// TIA Portal V17 export
// export: Created 2026-07-07T16:10:25.1870439Z, ExportSetting WithDefaults, DisplayName Totally Integrated Automation Portal, DisplayVersion V17, DisplayName TIA Portal Openness, DisplayVersion V17, DisplayName TIA Portal Version Control Interface, DisplayVersion V17, DisplayName STEP 7 Professional, DisplayVersion V17, DisplayName STEP 7 Safety, DisplayVersion V17, DisplayName WinCC Professional, DisplayVersion V17
FUNCTION_BLOCK "Manchester_Decoding"   // FB2, LAD
{ S7_Optimized_Access := 'TRUE' }
VERSION : 0.1
// stored: AutoNumber true, IsIECCheckEnabled false, IsRetainMemResEnabled false, MemoryReserve 100, SetENOAutomatically false, UDAEnableTagReadback false
   VAR_INPUT
      Clock_signal : Bool;
      Data_signal : Bool;
      "No. of inputs" : Int;
      "Interchar_duration(ms)" : Int;
   END_VAR
   VAR_OUTPUT
      Input_1 : Bool;
      Input_2 : Bool;
      Input_3 : Bool;
      Input_4 : Bool;
      Input_5 : Bool;
      Input_6 : Bool;
      Input_7 : Bool;
      Input_8 : Bool;
   END_VAR
   VAR
      clock_begin : Bool;
      clock_end : Bool;
      clock_begin_pt : Time;
      duration_conv : Int;
      clock_begin_timer : IEC_TIMER;
   END_VAR
   VAR RETAIN
      clock_end_timer { S7_SetPoint := 'True'} : IEC_TIMER;
   END_VAR
   VAR
      clock_signal_counter { S7_SetPoint := 'True'} : IEC_COUNTER;
   END_VAR
BEGIN

REGION Network 1
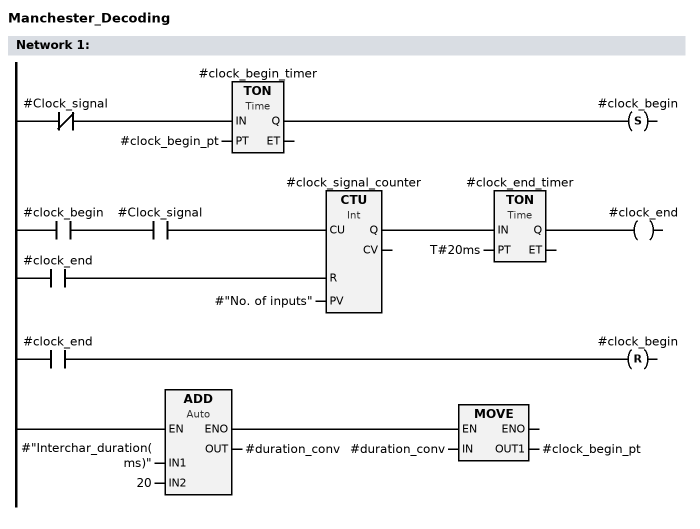
   RUNG wire#powerrail
      I_Contact( #Clock_signal )
      { S7_Templates := "time_type := Time" } #clock_begin_timer.TON(pt := #clock_begin_pt, et =>)
      S_Coil( #clock_begin )
   END_RUNG
   RUNG wire#powerrail
      Contact( #clock_begin )
      Contact( #Clock_signal )
      { S7_Templates := "value_type := Int" } #clock_signal_counter.CTU(r := wire#w1, pv := #"No. of inputs", cv =>)
      { S7_Templates := "time_type := Time" } #clock_end_timer.TON(pt := T#20ms, et =>)
      Coil( #clock_end )
   END_RUNG
   RUNG wire#powerrail
      Contact( #clock_end )
   END_RUNG wire#w1
   RUNG wire#powerrail
      Contact( #clock_end )
      R_Coil( #clock_begin )
   END_RUNG
   RUNG wire#powerrail
      Add(in1 := #"Interchar_duration(ms)", in2 := 20, out => #duration_conv)
      Move(in := #duration_conv, out1 => #clock_begin_pt)
   END_RUNG
   // the same network as SCL:
   #clock_begin_timer.TON(IN := NOT #Clock_signal, PT := #clock_begin_pt);
   IF #clock_begin_timer.Q THEN #clock_begin := TRUE; END_IF;
   #clock_signal_counter.CTU(CU := #clock_begin AND #Clock_signal, R := #clock_end, PV := #"No. of inputs");
   #clock_end_timer.TON(IN := #clock_signal_counter.Q, PT := T#20ms);
   #clock_end := #clock_end_timer.Q;
   IF #clock_end THEN #clock_begin := FALSE; END_IF;
   #duration_conv := #"Interchar_duration(ms)" + 20;
   #clock_begin_pt := #duration_conv;
END_REGION

REGION Network 2 (SCL)
   CASE #clock_signal_counter.CV OF
       1:
           #Input_1 := #Data_signal;
       2:
           #Input_2 := #Data_signal;
       3:
           #Input_3 := #Data_signal;
       4:
           #Input_4 := #Data_signal;
       5:
           #Input_5 := #Data_signal;
       6:
           #Input_6 := #Data_signal;
       7:
           #Input_7 := #Data_signal;
       8:
           #Input_8 := #Data_signal;
   END_CASE;
END_REGION
END_FUNCTION_BLOCK
